PROGRAM MAIN
VAR
	insertion : PneumaticInsertion;
	
	enable : BOOL;
	up : BOOL;
	down : BOOL;
	
	in : BOOL;
	out : BOOL;
	
	suction : ARRAY[1..4] OF SuctionPad;
	enableAllSuction : BOOL;
	i : INT;
END_VAR

insertion(
	enable:= enable, 
	slider=> , 
	screw=> , 
	contact=> , 
	home=> , 
	ready=> , 
	busy=> , 
	error=> , 
	homeSet=> );

IF NOT insertion.homeSet THEN
	insertion.homingSequence();
	RETURN;
END_IF

insertion.stop();
	
IF in THEN
	insertion.press();
	out := FALSE;
END_IF

IF out THEN
	insertion.release();
	in := FALSE;
END_IF

IF up THEN
	insertion.slideContinuous(direction:= MC_Positive_Direction);
	down := FALSE;
END_IF

IF down THEN
	insertion.slideContinuous(direction:= MC_Negative_Direction);
	up := FALSE;
END_IF

IF enableAllSuction THEN
	FOR i:=1 TO 4 BY 1 DO
		suction[i].enable := TRUE;
	END_FOR
END_IF

END_PROGRAM

(* stored: Version 1.1.0.1, ProductVersion 3.1.4024.11
   POU MAIN: Id {44291347-8ac8-42fe-bc2b-4cb56be25214}, SpecialFunc None *)
